(* IEC 61131-3 sources: SIGMATEK-Jumag-Utils-Examples/functionTrigger/Class/Class0, 1 file *)

(* ---- Class0.st ---- *)
(*!
<Class
	Name               = "Class0"
	Revision           = "0.0"
	RealtimeTask       = "false"
	CyclicTask         = "true"
	DefCyclictime      = "100 ms"
	BackgroundTask     = "false"
	Sigmatek           = "false"
	OSInterface        = "false"
	HighPriority       = "false"
	Automatic          = "false"
	UpdateMode         = "Prescan"
	SharedCommandTable = "true"
	Objectsize         = "(284,120)">
	<Channels>
		<Server Name="ClassSvr" Visualized="false" Initialize="false" WriteProtected="true" Retentive="false"/>
		<Server Name="qBlink" Visualized="false" Initialize="false" WriteProtected="true" Retentive="false"/>
		<Server Name="targetTime" Visualized="false" Initialize="true" DefValue="1000" WriteProtected="false" Retentive="false"/>
	</Channels>
	<Dependencies>
		<Files>
			<File Path=".\Source\functionTrigger.c"/>
		</Files>
	</Dependencies>
</Class>
*)
Class0 : CLASS
  //Servers:
	ClassSvr 	: SvrChCmd_DINT;
	targetTime 	: SvrCh_UDINT;
	qBlink 	: SvrCh_DINT;
  //Clients:
  //Variables:
  //Functions:

	FUNCTION VIRTUAL GLOBAL CyWork
		VAR_INPUT
			EAX 	: UDINT;
		END_VAR
		VAR_OUTPUT
			state (EAX) 	: UDINT;
		END_VAR;

	FUNCTION state
		VAR_OUTPUT
			ret_code 	: ConfStates;
		END_VAR;
  //Tables:
	FUNCTION @STD
		VAR_OUTPUT
			ret_code	: CONFSTATES;
		END_VAR;
	FUNCTION GLOBAL TAB @CT_;
END_CLASS;

// Declaration of C Function
Function Global __cdecl functionTrigger
VAR_INPUT
  CURR_TIME : UDINT;
  TIME_STAMP : ^UDINT;
  TAR_TIME : UDINT;
END_VAR
VAR_OUTPUT
  Q : BOOL;
END_VAR;

FUNCTION VIRTUAL GLOBAL Class0::CyWork
	VAR_INPUT
		EAX 	: UDINT;
	END_VAR
	VAR_OUTPUT
		state (EAX) 	: UDINT;
	END_VAR
  VAR
  	functionTimeStamp : ^UDINT;
  END_VAR

  if (functionTrigger(CURR_TIME := ops.tAbsolute, TIME_STAMP := functionTimeStamp, TAR_TIME := 1000)) then
    qblink := true;
  else
    qBlink := false;
  end_if;

	state := READY;

END_FUNCTION
